FUNCTION_BLOCK Composite
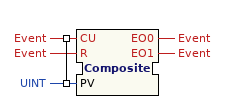
  EVENT_INPUT
    CU WITH PV;
    R;
  END_EVENT
  EVENT_OUTPUT
    EO0;
    EO1;
  END_EVENT
  VAR_INPUT
    PV : UINT := 0;
  END_VAR
  FBS
    E_CTU_CUSTOM : E_CTU_CUSTOM;
    E_SWITCH_CUSTOM : E_SWITCH_CUSTOM;
    CvToGTranslator : CvToGTranslator;
  END_FBS
  EVENT_CONNECTIONS
    E_CTU_CUSTOM.CUO TO E_SWITCH_CUSTOM.EI;
    CU TO E_CTU_CUSTOM.CU;
    E_SWITCH_CUSTOM.EO0 TO EO0;
    E_SWITCH_CUSTOM.EO1 TO EO1;
    R TO E_CTU_CUSTOM.R;
  END_CONNECTIONS
  DATA_CONNECTIONS
    PV TO E_CTU_CUSTOM.PV;
    E_CTU_CUSTOM.CV TO CvToGTranslator.CV;
    CvToGTranslator.G TO E_SWITCH_CUSTOM.G;
  END_CONNECTIONS
END_FUNCTION_BLOCK
